(* CODESYS project S7Comm.library
   Author: 夏远飞
   Version: 1.0.0.0
   Title: S7Comm
   Company: 赛克华石

Project tree, tasks and I/O mapping:
  libraries: Standard, * (System); Network, 3.5.7.0 (3S - Smart Software Solutions GmbH)
  function block TCP客户端 [ST]
  function block S7Comm [ST]
*)

// TCP客户端
FUNCTION_BLOCK TCP客户端
VAR_INPUT
	IP地址:STRING;
	端口号:UINT;
	发送:BOOL;
	发送字节数:INT;
	发送区指针:POINTER TO BYTE;
	接收字节数:INT;
	接收区指针:POINTER TO BYTE;	
END_VAR
VAR_OUTPUT
	连接成功:BOOL;
	发送完成:BOOL;
	接收终止:BOOL;
	接收成功:BOOL;
	实际接收数:ULINT;
	xError:BOOL;
	eError: NBS.ERROR;
END_VAR
VAR
	ipAddr:NBS.IP_ADDR;
	TCP_Client_0: NBS.TCP_Client;
	TCP_Read_0: NBS.TCP_Read;
	TCP_Write_0: NBS.TCP_Write;	
	TON_0: TON;
END_VAR

ipAddr.sAddr:= IP地址;
TON_0(IN:= TCP_Client_0.xDone OR TCP_Client_0.xError OR TCP_Read_0.xError OR TCP_Write_0.xError , PT:= T#200MS, Q=> , ET=> );
TCP_Client_0(
	xEnable:= NOT TON_0.Q, 
	xDone=> , 
	xBusy=> , 
	xError=> , 
	udiTimeOut:= 1000000, 
	ipAddr:= ipAddr, 
	uiPort:= 端口号, 
	eError=> , 
	xActive=> 连接成功, 
	hConnection=> );
IF 接收字节数 = 0 THEN
	接收字节数 := 80;
END_IF
TCP_Read_0(
	xEnable:= TCP_Client_0.xActive, 
	xDone=> 接收终止, 
	xBusy=> , 
	xError=> , 
	hConnection:= TCP_Client_0.hConnection, 
	szSize:= INT_TO_UINT(接收字节数), 
	pData:= 接收区指针, 
	eError=> , 
	xReady=> 接收成功, 
	szCount=> );
TCP_Write_0(
	xExecute:= 发送, 
	udiTimeOut:= 500000, 
	xDone=> 发送完成, 
	xBusy=> , 
	xError=> , 
	hConnection:= TCP_Client_0.hConnection, 
	szSize:= INT_TO_UINT(发送字节数), 
	pData:= 发送区指针, 
	eError=> );
IF TCP_Client_0.xError THEN
	eError := TCP_Client_0.eError;
END_IF
IF TCP_Read_0.xError THEN
	eError := TCP_Read_0.eError;
END_IF
IF TCP_Write_0.xError THEN
	eError := TCP_Write_0.eError;
END_IF
IF TCP_Read_0.xReady THEN
	实际接收数 := TCP_Read_0.szCount;
END_IF
xError := TCP_Client_0.xError OR TCP_Read_0.xError OR TCP_Write_0.xError;
IF NOT xError THEN
	eError := 0;
END_IF

END_FUNCTION_BLOCK

// S7Comm
FUNCTION_BLOCK S7Comm
VAR_INPUT
	IP地址			:STRING;
	数据读取指针	:POINTER TO BYTE;
	读取长度		:UINT (0..200);
	读取DB号		:UINT;
	读地址偏移		:UINT;
	数据发送指针	:POINTER TO BYTE;
	发送长度		:UINT (0..200);
	发送DB号		:UINT;
	写地址偏移		:UINT;
END_VAR
VAR_OUTPUT
	连接状态	:INT;
	数据包		:UINT;
	包每秒		:UINT;
	读取成功	:BOOL;
	读取计数	:UDINT;
	读取出错	:BOOL;
	写入成功	:BOOL;
	写入计数	:UDINT;
	写入出错	:BOOL;
END_VAR
VAR
	TCP客户端_0:TCP客户端;
	发送包:ARRAY[0..255] OF BYTE;
	发送包长度:INT;
	发送请求:BOOL;
	发送完成:BOOL;
	接收包:ARRAY[0..255] OF BYTE;
	接收包长度:INT;
	接收成功:BOOL;
	pt:POINTER TO BYTE;
	i :INT;
	最大长度:INT;
	连接成功P: R_TRIG;
	数据包自加P: R_TRIG;
	读取成功P: R_TRIG;
	写入成功P: R_TRIG;
	包每秒T: TON;
	上秒包数:UINT;
END_VAR

TCP客户端_0(
	IP地址:= IP地址, 
	端口号:= 102, 
	发送:= 发送请求, 
	发送字节数:= 发送包长度, 
	发送区指针:= ADR(发送包), 
	接收字节数:= 255, 
	接收区指针:= ADR(接收包), 
	连接成功=> , 
	发送完成=> 发送完成, 
	接收终止=> , 
	接收成功=> 接收成功, 
	实际接收数=> , 
	xError=> , 
	eError=> );

连接成功P(CLK:= TCP客户端_0.连接成功, Q=> );
IF 连接成功P.Q THEN
    连接状态:=1;
END_IF

IF 连接状态 =1 THEN		//握手包
	发送包[0]  := 16#03;//TPKT_Version	版本号
	发送包[1]  := 16#00;//TPKT_Reserved	预留
	发送包[2]  := 16#00;//TPKT_Length	长度
	发送包[3]  := 16#16;//TPKT_Length	长度
	发送包[4]  := 16#11;//COTP_Length	长度
	发送包[5]  := 16#E0;//COTP_Type		PDU类型		0xe0 CR 连接请求	0xd0 CC 连接确认	0xf0 数据传输
	发送包[6]  := 16#00;//COTP_DST_Ref	目标引用
	发送包[7]  := 16#00;//COTP_DST_Ref	目标引用
	发送包[8]  := 16#00;//COTP_SRC_Ref	源引用
	发送包[9]  := 16#01;//COTP_SRC_Ref	源引用
	发送包[10] := 16#00;//COTP_Opt
	发送包[11] := 16#C1;//Parameter_code	src_tasp	上位机
	发送包[12] := 16#02;//Parameter_Length
	发送包[13] := 16#10;//Parameter_Data	01->PG	02->OP	03->单边	10->双边
	发送包[14] := 16#00;//Parameter_Data	机架插槽
	发送包[15] := 16#C2;//Parameter_code	 
	发送包[16] := 16#02;//Parameter_Length
	发送包[17] := 16#03;//Parameter_Data	 
	发送包[18] := 16#01;//Parameter_Data	 
	发送包[19] := 16#C0;//Parameter_code	 
	发送包[20] := 16#01;//Parameter_Length
	发送包[21] := 16#0A;//Parameter_Data
	发送包长度	:= 22;
	发送请求	:= 1;
	IF 发送完成 THEN
		发送请求 := 0;
    	连接状态 := 2;
	END_IF
END_IF

IF 连接状态 = 2 AND 接收成功 THEN
	IF 接收包[5] = 16#D0 THEN
		连接状态 := 3;
	END_IF
END_IF

IF 连接状态 = 3 THEN	//通讯包
    发送包[0]  := 16#03;//TPKT_Version	版本号
	发送包[1]  := 16#00;//TPKT_Reserved	预留
	发送包[2]  := 16#00;//TPKT_Length	长度
	发送包[3]  := 16#19;//TPKT_Length	长度
	发送包[4]  := 16#02;//COTP_Length	长度
	发送包[5]  := 16#F0;//COTP_Type		PDU类型		0xe0 CR 连接请求	0xd0 CC 连接确认	0xf0 数据传输
	发送包[6]  := 16#80;//COTP_Opt
	发送包[7]  := 16#32;//协议ID
	发送包[8]  := 16#01;//0x01 Job Request主站发送请求  0x02 Ack 从站发送的简单确认  0x03 Ack-Data 带有可选数据字段的确认
	发送包[9]  := 16#00;//Reserved
	发送包[10] := 16#00;//Reserved
	发送包[11] := 16#00;//PDU Reference
	发送包[12] := 16#00;//PDU Reference
	发送包[13] := 16#00;//Parameter 参数长度	
	发送包[14] := 16#08;//Parameter 参数长度	
	发送包[15] := 16#00;//Data length 数据长度
	发送包[16] := 16#00;//Data length 数据长度
	发送包[17] := 16#F0;//功能码  设置通讯
	发送包[18] := 16#00;//Reserved
	发送包[19] := 16#00;// 
	发送包[20] := 16#01;//
	发送包[21] := 16#00;//
	发送包[22] := 16#01;// 
	发送包[23] := 16#03;//PDU长度
	发送包[24] := 16#C0;//PDU长度	
	发送包长度	:= 25;
	发送请求	:= 1;
	IF 发送完成 THEN
		发送请求 := 0;
    	连接状态 := 4;
	END_IF
END_IF

IF 连接状态 = 4 AND 接收成功 THEN
	IF 接收包[8] = 16#02 OR 接收包[8] = 16#03 THEN
		连接状态 := 5;
		最大长度 := SHL(TO_INT(接收包[25]),8) + TO_INT(接收包[26]);
	END_IF
END_IF

IF 连接状态 = 5 AND 读取长度 = 0 AND 发送长度 > 0 THEN
	连接状态 := 7;
END_IF
IF 连接状态 = 5 AND 读取长度 > 0 THEN	//读取数据
	读取成功 := 0;
    发送包[0]  := 16#03;//TPKT_Version	版本号
	发送包[1]  := 16#00;//TPKT_Reserved	预留
	发送包[2]  := 16#00;//TPKT_Length	长度
	发送包[3]  := 16#1F;//TPKT_Length	长度
	发送包[4]  := 16#02;//COTP_Length	长度
	发送包[5]  := 16#F0;//COTP_Type		PDU类型		0xe0 CR 连接请求	0xd0 CC 连接确认	0xf0 数据传输
	发送包[6]  := 16#80;//COTP_Opt
	发送包[7]  := 16#32;//协议ID
	发送包[8]  := 16#01;//0x01 Job Request主站发送请求  0x02 Ack 从站发送的简单确认  0x03 Ack-Data 带有可选数据字段的确认
	发送包[9]  := 16#00;//Reserved
	发送包[10] := 16#00;//Reserved
	发送包[11] := TO_BYTE(SHR(数据包,8) AND 16#FF);//PDU Reference
	发送包[12] := TO_BYTE(数据包 AND 16#FF);//PDU Reference
	发送包[13] := 16#00;//Parameter 参数长度
	发送包[14] := 16#0E;//Parameter 参数长度
	发送包[15] := 16#00;//Data length 数据长度
	发送包[16] := 16#00;//Data length 数据长度
	发送包[17] := 16#04;//功能码  读取数据
	发送包[18] := 16#01;//通讯项数
	发送包[19] := 16#12;//item1
	发送包[20] := 16#0A;//此字节往后的字节长度
	发送包[21] := 16#10;//指针地址格式
	发送包[22] := 16#02;//0x01 BOOL    0x02 BYTE    0x03 CHAR    0x04 WORD..........
	发送包[23] := TO_BYTE(SHR(读取长度,8) AND 16#FF);//数据长度
	发送包[24] := TO_BYTE(读取长度 AND 16#FF);//数据长度
	发送包[25] := TO_BYTE(SHR(读取DB号,8) AND 16#FF);//数据块号
	发送包[26] := TO_BYTE(读取DB号 AND 16#FF);//数据块号
	IF 读取DB号 = 0 THEN
		发送包[27] := 16#83;//81 in    82 out    83 M    84 DB........;
	ELSE
		发送包[27] := 16#84;//81 in    82 out    83 M    84 DB........;;
	END_IF
	发送包[28] := TO_BYTE(SHR(读地址偏移,11) AND 16#FF);//地址偏移
	发送包[29] := TO_BYTE(SHR(读地址偏移,5) AND 16#FF);//地址偏移
	发送包[30] := TO_BYTE(SHL(读地址偏移,3) AND 16#F8);//地址偏移
	发送包长度	:= 31;
	发送请求	:= 1;
	IF 发送完成 THEN
		发送请求 := 0;
    	连接状态 := 6;
	END_IF
END_IF
IF 连接状态 = 6 AND 接收成功 THEN
	IF 接收包[8] = 16#02 OR 接收包[8] = 16#03 THEN
		IF 接收包[21] = 16#FF THEN
			读取成功 := 1;
			读取出错 := 0;
    		pt := 数据读取指针;
			FOR i:=0 TO TO_INT(读取长度-1) BY 1 DO
    			pt^ := 接收包[25+i];
				pt := pt + 1;
			END_FOR
		ELSE
			读取出错 := 1;
		END_IF

		IF 发送长度 > 0 THEN
			连接状态 := 7;
		ELSE
    		连接状态 := 5;
		END_IF
	END_IF
END_IF

IF 连接状态 = 7 AND 发送长度 > 0 THEN	//发送数据
	写入成功 := 0;
    发送包[0]  := 16#03;//TPKT_Version	版本号
	发送包[1]  := 16#00;//TPKT_Reserved	预留
	发送包[2]  := TO_BYTE(SHR((35 + 发送长度),8) AND 16#FF);//TPKT_Length	长度
	发送包[3]  := TO_BYTE((35 + 发送长度) AND 16#FF);//TPKT_Length	长度
	发送包[4]  := 16#02;//COTP_Length	长度
	发送包[5]  := 16#F0;//COTP_Type		PDU类型		0xe0 CR 连接请求	0xd0 CC 连接确认	0xf0 数据传输
	发送包[6]  := 16#80;//COTP_Opt
	发送包[7]  := 16#32;//协议ID
	发送包[8]  := 16#01;//0x01 Job Request主站发送请求  0x02 Ack 从站发送的简单确认  0x03 Ack-Data 带有可选数据字段的确认
	发送包[9]  := 16#00;//Reserved
	发送包[10] := 16#00;//Reserved
	发送包[11] := TO_BYTE(SHR(数据包,8) AND 16#FF);//PDU Reference
	发送包[12] := TO_BYTE(数据包 AND 16#FF);//PDU Reference
	发送包[13] := 16#00;//Parameter 参数长度
	发送包[14] := 16#0E;//Parameter 参数长度
	发送包[15] := TO_BYTE(SHR((发送长度 + 4),8) AND 16#FF);//Data length 数据长度
	发送包[16] := TO_BYTE((发送长度 + 4) AND 16#FF);//Data length 数据长度
	发送包[17] := 16#05;//功能码  发送数据
	发送包[18] := 16#01;//通讯项数
	发送包[19] := 16#12;//item1
	发送包[20] := 16#0A;//此字节往后的字节长度
	发送包[21] := 16#10;//指针地址格式
	发送包[22] := 16#02;//0x01 BOOL    0x02 BYTE    0x03 CHAR    0x04 WORD.......
	发送包[23] := TO_BYTE(SHR(发送长度,8) AND 16#FF);	//数据长度
	发送包[24] := TO_BYTE(发送长度 AND 16#FF);			//数据长度
	发送包[25] := TO_BYTE(SHR(发送DB号,8) AND 16#FF);	//数据块号
	发送包[26] := TO_BYTE(发送DB号 AND 16#FF);			//数据块号
	IF 发送DB号 = 0 THEN
		发送包[27] := 16#83;//81 in    82 out    83 M    84 DB......
	ELSE
		发送包[27] := 16#84;//81 in    82 out    83 M    84 DB......
	END_IF
	发送包[28] := TO_BYTE(SHR(写地址偏移,11) AND 16#FF);	//地址偏移
	发送包[29] := TO_BYTE(SHR(写地址偏移,5) AND 16#FF);	//地址偏移
	发送包[30] := TO_BYTE(SHL(写地址偏移,3) AND 16#F8);	//地址偏移
	//item0
	发送包[31] := 16#00;
	发送包[32] := 16#04;//0x04  BYTE/WORD/DWORD    0x03 BIT    0x07 REAL......
	发送包[33] := TO_BYTE(SHR(发送长度,5) AND 16#FF);	//数据长度bit
	发送包[34] := TO_BYTE(SHL(发送长度,3) AND 16#F8);	//数据长度bit
	pt := 数据发送指针;
	FOR i:=0 TO TO_INT(发送长度-1) BY 1 DO
    	发送包[35+i] := pt^;
		pt := pt + 1;
	END_FOR
	发送包长度	:= 35 + TO_INT(发送长度);
	发送请求	:= 1;
	IF 发送完成 THEN
		发送请求 := 0;
    	连接状态 := 8;
	END_IF
END_IF

IF 连接状态 = 8 AND 接收成功 THEN
    IF 接收包[8] = 16#02 OR 接收包[8] = 16#03 THEN
		IF 接收包[21] = 16#FF THEN
    		写入成功 := 1;
			写入出错 := 0;
		ELSE
			写入出错 := 1;
		END_IF
		IF 读取长度 > 0 THEN
			连接状态 := 5;
		ELSE
    		连接状态 := 7;
		END_IF
	END_IF
END_IF

数据包自加P(CLK:= 连接状态 = 5 OR 连接状态 = 7, Q=> );
IF 数据包自加P.Q THEN
    数据包 := 数据包 + 1;
END_IF

包每秒T(IN:= NOT 包每秒T.Q, PT:= T#1S, Q=> , ET=> );
IF 包每秒T.Q THEN
	包每秒 := 数据包 - 上秒包数;
    上秒包数 := 数据包;
END_IF
读取成功P(CLK:= 读取成功, Q=> );
IF 读取成功P.Q THEN
    读取计数 := 读取计数 +1;
END_IF
写入成功P(CLK:= 写入成功, Q=> );
IF 写入成功P.Q THEN
    写入计数 := 写入计数 + 1;
END_IF

END_FUNCTION_BLOCK
